FUNCTION max_abs_array : LREAL
VAR_IN_OUT
	aData : ARRAY[*] OF LREAL;
END_VAR
VAR
	nIdx: DINT;
END_VAR

max_abs_array := 0;
FOR nIdx := LOWER_BOUND(aData,1) TO UPPER_BOUND(aData,1) DO
	max_abs_array := MAX(ABS(aData[nIdx]),max_abs_array);
END_FOR

END_FUNCTION

(* stored: Version 1.1.0.1, ProductVersion 3.1.4024.12
   POU max_abs_array: Id {09302b30-6778-4f22-a27d-96350aa85cf1}, SpecialFunc None *)
